PROGRAM Kommunikation_Client
VAR
	Connect			:FB_SocketConnect;
	Send			:FB_SocketSend;
	Receive 		:FB_SocketReceive;
	CloseAll		:FB_SocketCloseAll;
	
	sSrvNetId   : T_AmsNetId := '';
    sRemoteHost : T_IPv4Addr := '192.168.50.100';
    nRemotePort : UDINT := 30003;
    bConnect    : BOOL;
    tTimeout    : TIME := T#45S;(*!!!*)
	bSend		:BOOL;
	bReceive	:BOOL;
	
	hSocket    : T_HSOCKET;
	
	{attribute 'TcEncoding':='UTF-8'}
	//test		:T_MaxString := 'movej([0,1.57,-1.57,3.14,-1.57,1.57],a=0.2,v=0.2,t=0,r=0)/n'; 
	test		:T_MaxString := 'force()'; 
	{attribute 'TcEncoding':='UTF-8'}
	Test2		:STRING := 'socket_send_byte(10)'; 
	test6		:ARRAY[0..7] OF BYTE := [102,111,114,99,101,40,41,10];

	
END_VAR

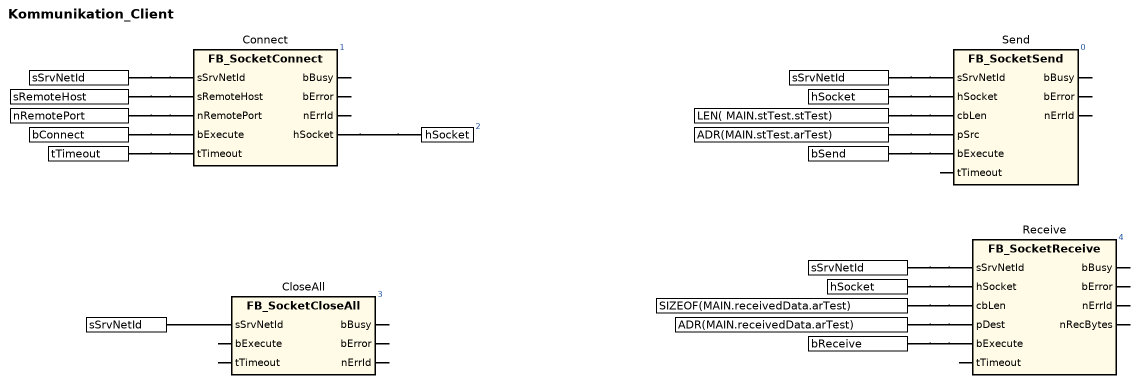
Send(
    sSrvNetId := sSrvNetId,
    hSocket := hSocket,
    cbLen := LEN( MAIN.stTest.stTest),
    pSrc := ADR(MAIN.stTest.arTest),
    bExecute := bSend); // FB_SocketSend
Connect(
    sSrvNetId := sSrvNetId,
    sRemoteHost := sRemoteHost,
    nRemotePort := nRemotePort,
    bExecute := bConnect,
    tTimeout := tTimeout); // FB_SocketConnect
hSocket := Connect.hSocket;
CloseAll(sSrvNetId := sSrvNetId); // FB_SocketCloseAll
Receive(
    sSrvNetId := sSrvNetId,
    hSocket := hSocket,
    cbLen := SIZEOF(MAIN.receivedData.arTest),
    pDest := ADR(MAIN.receivedData.arTest),
    bExecute := bReceive); // FB_SocketReceive

END_PROGRAM

(* stored: Version 1.1.0.1
   POU Kommunikation_Client: Id {1cdd5e72-6f0a-405e-91e1-56fefb5cfbd9}, SpecialFunc None *)
